// TIA Portal project "SCDW_TEST_36d450a4" (V17)

(* hardware
DEVICE "SCDW_TEST_PLC"  S7-1200 Station
   slot 0: "Rack_0"  S7-1200 Rack  Rack  V1.0
   slot 1: "SCDW_TEST_PLC"  CPU 1214C AC/DC/Rly  6ES7 214-1BG40-0XB0  V4.4
*)

// ===== PLC "SCDW_TEST_PLC"  CPU 1214C AC/DC/Rly =====

DATA_BLOCK "SCDW_STEP3_IDB"   // DB0
{ S7_Optimized_Access := 'TRUE' }
VERSION : 0.1
// stored: InstanceOfName SCDW_STEP3_FB
"SCDW_STEP3_FB"
BEGIN
END_DATA_BLOCK

FUNCTION_BLOCK "SCDW_STEP3_FB"   // FB1, LAD
{ S7_Optimized_Access := 'TRUE' }
   VAR
      State : Bool;
   END_VAR
BEGIN

REGION Network 1: 状态保持
   // 辅助FB状态程序段。
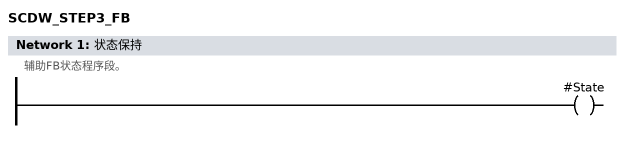
   RUNG wire#powerrail
      Coil( #State )
   END_RUNG
   // the same network as SCL:
   #State := TRUE;
END_REGION
END_FUNCTION_BLOCK

FUNCTION "SCDW_STEP3_FC" : Void   // FC1, LAD
{ S7_Optimized_Access := 'TRUE' }
   VAR_TEMP
      Dummy : Bool;
   END_VAR
BEGIN

REGION Network 1: 调用辅助FB
   // 使用真实背景DB调用辅助FB。
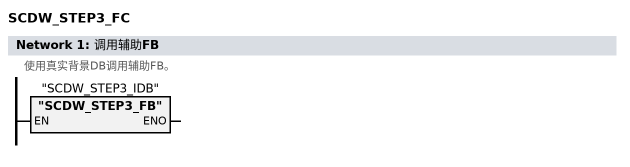
   RUNG wire#powerrail
      "SCDW_STEP3_IDB"()
   END_RUNG
   // the same network as SCL:
   "SCDW_STEP3_IDB"();   // "SCDW_STEP3_FB"
END_REGION
END_FUNCTION

ORGANIZATION_BLOCK "Main"   // OB1, LAD, ProgramCycle
TITLE = "Main Program Sweep (Cycle)"
{ S7_Optimized_Access := 'TRUE' }
VERSION : 0.1
   VAR_INPUT
      Initial_Call : Bool;   // Initial call of this OB
      Remanence : Bool;   // =True, if remanent data are available
   END_VAR
BEGIN
END_ORGANIZATION_BLOCK